// TIA Portal V20 export
DATA_BLOCK "CallEquipment_DB"   // DB140
{ DB_Accessible_From_OPC_UA := 'FALSE' }
// stored: AssignedProDiagFB Unit1.Em0.ProDiag, DBAccessibleFromOPCUA false, DBAccessibleFromWebserver false, InstanceOfName Unit1.Em0.CallEquipment, InstanceOfType FB, Namespace Unit1.Em0
"Unit1.Em0.CallEquipment"
   // VAR_INPUT
   //    ZoneOperationEnable { ExternalWritable := 'False'} : "LWONIK_typeSafetyZoneManualOperation";
   // END_VAR
   // VAR_IN_OUT
   //    unitStatus : "LAF_typeUnitStatus";
   //    emFeedback : "LUC_typeEmFeedback";
   //    unitAlarmDB : "LAF_typeAlarms";
   // END_VAR
   // VAR
   //    InstStacker1NgBoxSequence { ExternalWritable := 'False'} : "Unit1.Em0.Sequence_1_Stacker1NgBox";
   //    instStacker1NgBoxHomeJob1 { ExternalWritable := 'False'} : "LAF_SelectJob";
   //    instStacker1NgBoxLoadJob2 { ExternalWritable := 'False'} : "LAF_SelectJob";
   //    instStacker1NgBoxUnloadJob3 { ExternalWritable := 'False'} : "LAF_SelectJob";
   //    instCmStacker1NgBoxFullDetect { ExternalWritable := 'False'} : "LBC_DigitalSignalCn";
   //    instCmStacker1NgBoxDetect { ExternalWritable := 'False'} : "LBC_DigitalSignalCn";
   //    instCmStacker1NgBoxLoadingUpDown { ExternalWritable := 'False'} : "LBC_TwoWayActuatorCn";
   //    instCmStacker1NgBoxUnitMoverBwdFwd { ExternalWritable := 'False'} : "LBC_TwoWayActuatorCn";
   //    instCmStacker1NgBoxClampLeftOpenClose { ExternalWritable := 'False'} : "LBC_TwoWayActuatorCn";
   //    instCmStacker1NgBoxClampRightOpenClose { ExternalWritable := 'False'} : "LBC_TwoWayActuatorCn";
   //    instCmStacker1NgBoxClampMoverOpenClose { ExternalWritable := 'False'} : "LBC_TwoWayActuatorCn";
   //    instCmStacker1NgBoxLiftDownUp { ExternalWritable := 'False'} : "LBC_TwoWayActuatorCn";
   //    instCmStacker1NgBoxLockDownUp { ExternalWritable := 'False'} : "LBC_TwoWayActuatorCn";
   //    instManageAlarms { ExternalWritable := 'False'} : "LAF_ManageAlarms";
   //    instEventsPFE { ExternalWritable := 'False'} : "Unit1.Em0.EventsPFE";
   //    statUnitStatus { ExternalWritable := 'False'} : "LAF_typeUnitStatus";
   //    statTonTime { ExternalWritable := 'False'} : Array[0..999] of TON_TIME;
   //    statTofTime { ExternalWritable := 'False'} : Array[0..99] of TOF_TIME;
   //    statPulse { ExternalWritable := 'False'} : Array[0..999] of Bool;
   //    statEnableManualCmds { ExternalWritable := 'False'} : Bool;
   //    "*** Interlock TwoWay ***" { S7_SetPoint := 'True'} : "LER_Axis_Homing";
   //    instCmStacker1NgBoxLoadingUpDownInterlock { S7_SetPoint := 'True'} : Array[0..2] of "LER_Actuator";
   //    instCmStacker1NgBoxUnitMoverBwdFwdInterlock { S7_SetPoint := 'True'} : Array[0..2] of "LER_Actuator";
   //    instCmStacker1NgBoxClampLeftOpenCloseInterlock { S7_SetPoint := 'True'} : Array[0..2] of "LER_Actuator";
   //    instCmStacker1NgBoxClampRightOpenCloseInterlock { S7_SetPoint := 'True'} : Array[0..2] of "LER_Actuator";
   //    instCmStacker1NgBoxClampMoverOpenCloseInterlock { S7_SetPoint := 'True'} : Array[0..2] of "LER_Actuator";
   //    instCmStacker1NgBoxLiftDownUpInterlock { S7_SetPoint := 'True'} : Array[0..2] of "LER_Actuator";
   //    instCmStacker1NgBoxLockDownUpInterlock { S7_SetPoint := 'True'} : Array[0..2] of "LER_Actuator";
   //    instCmStacker1NgBoxLoadingUpDown_IntPos : Array[0..2] of Struct
   //       "Int" : Array[1..10] of Bool;
   //    END_STRUCT;
   //    instCmStacker1NgBoxUnitMoverBwdFwd_IntPos : Array[0..2] of Struct
   //       "Int" : Array[1..10] of Bool;
   //    END_STRUCT;
   //    instCmStacker1NgBoxClampLeftOpenClose_IntPos : Array[0..2] of Struct
   //       "Int" : Array[1..10] of Bool;
   //    END_STRUCT;
   //    instCmStacker1NgBoxClampRightOpenClose_IntPos : Array[0..2] of Struct
   //       "Int" : Array[1..10] of Bool;
   //    END_STRUCT;
   //    instCmStacker1NgBoxClampMoverOpenClose_IntPos : Array[0..2] of Struct
   //       "Int" : Array[1..10] of Bool;
   //    END_STRUCT;
   //    instCmStacker1NgBoxLiftDownUp_IntPos : Array[0..2] of Struct
   //       "Int" : Array[1..10] of Bool;
   //    END_STRUCT;
   //    instCmStacker1NgBoxLockDownUp_IntPos : Array[0..2] of Struct
   //       "Int" : Array[1..10] of Bool;
   //    END_STRUCT;
   //    citi_Ptrig : Array[0..20] of Bool;
   //    citiTon : Array[0..20] of TON_TIME;
   //    citi : Time;
   //    citiTest : Array[0..20] of Bool;
   // END_VAR
BEGIN
   // instCmStacker1NgBoxLockDownUp.feedbackWorkPos : stack1NgBoxLockUp
END_DATA_BLOCK
